// TwinCAT 3 PLC project OpcUa_Lib
// Title: OpcUa_Lib
// Company: Chua Siang Poh
// Author: Chua Siang Poh
// ProjectVersion: 0.1.0
// ProgramVersion: 3.1.4020.10
// libraries:
//   Tc2_Standard, * (Beckhoff Automation GmbH)
//   Tc2_System, * (Beckhoff Automation GmbH)
//   Tc3_Module, * (Beckhoff Automation GmbH)
//   Tc3_PLCopen_OpcUa, * (Beckhoff Automation GmbH)
// project tree:
//   Base Component/OPC Client/ C_OPCCLIENT.TcPOU, GET_BECKHOFF_OPCUA_NAMESPACE.TcPOU (not stored), GET_OPCUA_SERVER_URL.TcPOU (not stored), S_UA_SERVERNAMESPACE.TcDUT
// (motion and I/O tree: see PLC project motion_library)
// real-time tasks:
//   TASK PlcTask: cycle T#10ms, priority 20, ADS port 350

// ---- Base Component/OPC Client/S_UA_SERVERNAMESPACE.TcDUT
TYPE S_UA_SERVERNAMESPACE :
STRUCT
	NAMESPACE 	: STRING(255);
	HANDLE		: UINT;
END_STRUCT
END_TYPE

// ---- Base Component/OPC Client/C_OPCCLIENT.TcPOU
FUNCTION_BLOCK C_OPCCLIENT
VAR_INPUT
END_VAR
VAR_OUTPUT
END_VAR
VAR
	_FBCONNECT 		: UA_Connect;
	_FBDISCONNECT 	: UA_Disconnect;
	_FBNAMESPACE	: UA_GetNamespaceIndex;
	_FBGETHANDLE	: UA_NodeGetHandle;
	_FBRELEASEHANDLE: UA_NodeReleaseHandle;
	_FBREAD 		: UA_Read;
	_FBWRITE 		: UA_Write;
	
	_HNDL			: DWORD;
	_SESSIONINFO	: ST_UASessionConnectInfo;
	_SERVERNAMESPACE: S_UA_SERVERNAMESPACE;
	
	_INTERNALSTATE 	: DINT;
	_NAMESPACEHANDLE: DWORD;
	_NAMESPACEARRAY	: ARRAY[0..15] OF STRING(255);
END_VAR

METHOD CONNECT : DINT
VAR_INPUT
	SERVER : STRING(255);
END_VAR
VAR
	NODE : ST_UANodeId;
END_VAR
IF _HNDL <> 0 THEN
	CONNECT := 1;
	RETURN;
END_IF

_SESSIONINFO.eSecurityMode := E_UASecurityMsgMode.eUASecurityMsgMode_None;
_SESSIONINFO.eSecurityPolicyUri := E_UASecurityPolicy.eUASecurityPolicy_None;
_SESSIONINFO.eTransportProfileUri := E_UATransportProfile.eUATransportProfileUri_UATcp;
_SESSIONINFO.tConnectTimeout := T#1M;
_SESSIONINFO.tSessionTimeout := T#1M;

_FBCONNECT(
	Execute:= TRUE, 
	ServerUrl:= SERVER, 
	SessionConnectInfo:= _SESSIONINFO, 
	Timeout:= , 
	ConnectionHdl=>  );
IF _FBCONNECT.Error THEN
	_FBCONNECT(Execute:= FALSE);
	CONNECT := 2;
	RETURN;
ELSIF _FBCONNECT.Done THEN
	_FBCONNECT(Execute:= FALSE);
	_HNDL := _FBCONNECT.ConnectionHdl;
	CONNECT := -1;
	RETURN;
ELSE
	CONNECT := 0;
	RETURN;
END_IF
END_METHOD

PROPERTY CONNECTED : BOOL
GET
CONNECTED := _HNDL <> 0;
END_GET
END_PROPERTY

METHOD DISCONNECT : DINT
VAR_INPUT
END_VAR
_FBDISCONNECT(
	Execute:= TRUE, 
	ConnectionHdl:= _HNDL, 
	Timeout:= , 
	Done=> , 
	Busy=> , 
	Error=> , 
	ErrorID=> );
IF _FBDISCONNECT.Error THEN
	_FBDISCONNECT(Execute:= FALSE);
	DISCONNECT := 1;
	RETURN;
ELSIF _FBDISCONNECT.Done THEN
	_HNDL := 0;
	_FBDISCONNECT(Execute:= FALSE);
	DISCONNECT := -1;
	RETURN;
ELSE
	DISCONNECT := 0;
	RETURN;
END_IF
END_METHOD

METHOD GENERATE_HANDLE : DINT
VAR_INPUT
	NAME 		: STRING(255);
	IS_NUMERIC_ID	: BOOL;
	HANDLE_PTR_OUT	: POINTER TO DWORD;
END_VAR
VAR
	NODE : ST_UANodeId;
END_VAR
IF HANDLE_PTR_OUT = 0 THEN
	GENERATE_HANDLE := 1;
	RETURN;
END_IF

IF IS_NUMERIC_ID THEN
	NODE.eIdentifierType := E_UAIdentifierType.eUAIdentifierType_Numeric;
ELSE
	NODE.eIdentifierType := E_UAIdentifierType.eUAIdentifierType_String;
END_IF
NODE.nNamespaceIndex := _SERVERNAMESPACE.HANDLE;
NODE.sIdentifier := NAME;

_FBGETHANDLE(
	Execute:= TRUE, 
	ConnectionHdl:= _HNDL, 
	NodeID:= NODE, 
	Timeout:= );
IF _FBGETHANDLE.Error THEN
	_FBGETHANDLE(Execute:= FALSE);
	GENERATE_HANDLE := 2;
	RETURN;
ELSIF _FBGETHANDLE.Done THEN
	HANDLE_PTR_OUT^ := _FBGETHANDLE.NodeHdl;
	_FBGETHANDLE(Execute:= FALSE);
	GENERATE_HANDLE := -1;
	RETURN;
ELSE
	GENERATE_HANDLE := 0;
	RETURN;
END_IF
END_METHOD

PROPERTY NAMESPACE : STRING(255)
GET
NAMESPACE := _SERVERNAMESPACE.NAMESPACE;
END_GET
END_PROPERTY

METHOD READ : DINT
VAR_INPUT
	HANDLE 			: DWORD;
	DATA_PTR_OUT	: PVOID;
	DATA_SIZE		: UDINT;
END_VAR
VAR
	ADDITIONAL_INFO	: ST_UANodeAdditionalInfo;
END_VAR
ADDITIONAL_INFO.nIndexRangeCount := 0;
ADDITIONAL_INFO.eAttributeID := E_UAAttributeID.eUAAI_Value;

_FBREAD(
	Execute:= TRUE, 
	ConnectionHdl:= _HNDL, 
	NodeHdl:= HANDLE, 
	stNodeAddInfo:= ADDITIONAL_INFO, 
	pVariable:= DATA_PTR_OUT, 
	cbData:= DATA_SIZE, 
	Timeout:= , 
	cbData_R=> );
IF _FBREAD.Error THEN
	_FBREAD(Execute:= FALSE); 
	READ := 1;
	RETURN;
ELSIF _FBREAD.Done THEN
	_FBREAD(Execute:= FALSE); 
	READ := -1;
	RETURN;
ELSE
	READ := 0;
	RETURN;
END_IF
END_METHOD

METHOD READ_RANGE : DINT
VAR_INPUT
	HANDLE 			: DWORD;
	START			: UDINT;
	END				: UDINT;
	DATA_PTR_OUT	: PVOID;
	DATA_SIZE		: UDINT;
END_VAR
VAR
	ADDITIONAL_INFO	: ST_UANodeAdditionalInfo;
END_VAR
ADDITIONAL_INFO.nIndexRangeCount := 1;
ADDITIONAL_INFO.eAttributeID := E_UAAttributeID.eUAAI_Value;
ADDITIONAL_INFO.stIndexRange[1].nStartIndex := START;
ADDITIONAL_INFO.stIndexRange[1].nEndIndex := END;

_FBREAD(
	Execute:= TRUE, 
	ConnectionHdl:= _HNDL, 
	NodeHdl:= HANDLE, 
	stNodeAddInfo:= ADDITIONAL_INFO, 
	pVariable:= DATA_PTR_OUT, 
	cbData:= DATA_SIZE, 
	Timeout:= , 
	cbData_R=> );
IF _FBREAD.Error THEN
	_FBREAD(Execute:= FALSE); 
	READ_RANGE := 1;
	RETURN;
ELSIF _FBREAD.Done THEN
	_FBREAD(Execute:= FALSE); 
	READ_RANGE := -1;
	RETURN;
ELSE
	READ_RANGE := 0;
	RETURN;
END_IF
END_METHOD

METHOD RELEASE_HANDLE : DINT
VAR_INPUT
	HANDLE : DWORD;
END_VAR
_FBRELEASEHANDLE(
	Execute:= TRUE, 
	ConnectionHdl:= _HNDL, 
	NodeHdl:= HANDLE, 
	Timeout:= , 
	Done=> , 
	Busy=> , 
	Error=> , 
	ErrorID=> );
IF _FBRELEASEHANDLE.Error THEN
	_FBRELEASEHANDLE(Execute:= FALSE);
	RELEASE_HANDLE := 1;
	RETURN;
ELSIF _FBRELEASEHANDLE.Done THEN
	_FBRELEASEHANDLE(Execute:= FALSE);
	RELEASE_HANDLE := -1;
	RETURN;
ELSE
	RELEASE_HANDLE := 0;
	RETURN;
END_IF
END_METHOD

METHOD RESOLVE_NAMESPACE : DINT
VAR_INPUT
	NAMESPACE : STRING(255);
END_VAR
_FBNAMESPACE(
	Execute:= TRUE, 
	ConnectionHdl:= _HNDL, 
	NamespaceUri:= NAMESPACE, 
	Timeout:= );
IF _FBNAMESPACE.Error THEN
	_FBNAMESPACE(Execute:= FALSE);
	RESOLVE_NAMESPACE := 1;
	RETURN;
ELSIF _FBNAMESPACE.Done THEN
	_SERVERNAMESPACE.NAMESPACE := NAMESPACE;
	_SERVERNAMESPACE.HANDLE := _FBNAMESPACE.NamespaceIndex;
	_FBNAMESPACE(Execute:= FALSE);
	RESOLVE_NAMESPACE := -1;
	RETURN;
ELSE
	RESOLVE_NAMESPACE := 0;
	RETURN;
END_IF
END_METHOD

END_FUNCTION_BLOCK
